
// ===== library: MasterCopy "DB_Diag_Com" =====

DATA_BLOCK "DB_Diag_Com"   // DB2
{ S7_Optimized_Access := 'FALSE' }
VERSION : 0.1
   VAR
      Ix_Debug_Bit : Array[0..15] of Bool;
      Ix_Debug_Int : Array[0..9] of Int;
      Ix_Debug_String : String[20];
      Qx_Debug_Bit : Array[0..15] of Bool;
      Qx_Debug_Int : Array[0..9] of Int;
      Qx_Debug_String : String[20];
   END_VAR
BEGIN
END_DATA_BLOCK